(* IEC 61131-3 sources: plc_on_fpga_riscv_hybrid/RV_FPGA_PLC_IDE_Projects/not, 1 file *)

(* ---- not.il ---- *)
VAR
END_VAR

PROGRAM not
    nn :
        LDN    %SW.0
        ST     %LEDR.0
END_PROGRAM
